FUNCTION Fakultaet : LINT
VAR_INPUT
	i_fakultat : INT;
END_VAR
VAR
	l_result : LINT := 1;
	i : INT;
END_VAR

FOR i := 1 TO i_fakultat BY 1 DO
	IF(i_fakultat = 0)
		THEN
		l_result := 1;
		RETURN;
	END_IF
l_result := l_result * i;
END_FOR;
Fakultaet := l_result;

END_FUNCTION

(* stored: Version 1.1.0.1, ProductVersion 3.1.4022.12
   POU Fakultaet: Id {5e87f3fe-03f9-42f4-97aa-37b27575a8c7}, SpecialFunc None *)
